(* PLC project EmergencyStopTest *)
(* stored: creationDateTime 2024-01-01T00:00:00, modificationDateTime 2024-01-01T00:00:00 *)

PROGRAM Main
  VAR
    X010 : BOOL;
    X001 : BOOL;
    Y001 : BOOL;
  END_VAR

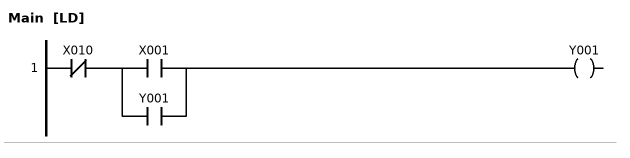
(* LD diagram, written out as Structured Text *)
Y001 := NOT X010 AND (X001 OR Y001);
END_PROGRAM

CONFIGURATION Config
  RESOURCE Res ON PLC
    TASK Main(INTERVAL := T#20ms, PRIORITY := 0);
    PROGRAM Main WITH Main : Main;
  END_RESOURCE
END_CONFIGURATION
